(* Schneider Machine Expert - Basic project ECC, file version 2.0.0.0 *)
(* ProjectInformations: Name=New project *)

HARDWARE
  Cpu 0: TM221CE16T
  Cartridge1 0: TMC2SL1
  EthernetConfiguration: NetworkName=M221, IpAllocationMode=FixedAddress, IpAddress=192.168.1.10, SubnetMask=255.255.255.0
  EthernetConfiguration: NetworkName=M221, IpAllocationMode=FixedAddress, IpAddress=0.0.0.0, SubnetMask=0.0.0.0
  SerialLineConfiguration: Baud=Baud9600, Parity=ParityNone, DataBits=DataBits8, StopBits=StopBits1, PhysicalMedium=PhysicalMediumRs485, TransmissionMode=TransmissionModeModbusRtu, SlaveId=1, Addressing=MasterAddressing
  MastTask: UsePeriodScanMode=false, PeriodScan=100
  FastTask: Period=255
  CpuBehavior: StartingMode=StartAsPreviousState, AutoSaveRamOnEeprom=true, WatchdogPeriod=250

SYMBOLS  (address, symbol, comment, settings)
  %MW5:X2   BUZZER
  %MW5:X3   FLICKER
  %M100       "机械报警&蜂鸣器接口"
  %M103       "报警闪烁接口"
  %M110       "主机主滑油进口压力过低降速输出"
  %M111       "主机滑油进口温度过高降速输出"
  %M112       "主机十字头滑油进口压力过低降速输出"
  %M113       "主机推力轴承油温度过高降速输出"
  %M120       "主机增压器滑油进口压力过低降速输出"
  %M121       "主机增压器滑油出口温度过高降速输出"
  %M122       "主机缸套冷却水进口压力过低降速输出"
  %M129       "主机空气弹簧气源进口压力过低降速输出"
  %M130       "主机空冷器后扫气温度过高降速输出"
  %M131       "主机增压器前排气温度过高降速输出"
  %M132       "主机增压器后排气温度过高降速输出"
  %M200       "原先是%M100"
  %S5       SB_TB100MS  "内部时钟生成的 100 毫秒时基"
  %MW4        "通讯故障"
  %TM0        "可修改通讯间隔，默认10ms"  [Preset=10, Base=TenMilliSeconds]
  %TM1        [Preset=5, Base=OneHundredMilliSeconds]
  %TM2        [Preset=5, Base=OneHundredMilliSeconds]
  %TM3        [Preset=15, Base=OneSecond]
  %READ_VAR0   [Link(Value(FBComLinkParameterEnums=SerialLine1)), RemoteDeviceId(Value(int=1)), Timeout(Value(int=3)), ObjType(Value(FBComObjTypeParameterEnums=IW)), FirstObj(Value(int=513)), Quantity(Value(int=4)), IndexData(Value(int=0))]
  %WRITE_VAR0   [Link(Value(FBComLinkParameterEnums=SerialLine1)), RemoteDeviceId(Value(int=2)), Timeout(Value(int=3)), ObjType(Value(FBComObjTypeParameterEnums=MW)), FirstObj(Value(int=513)), Quantity(Value(int=2)), IndexData(Value(int=5))]
  %WRITE_VAR1   [Link(Value(FBComLinkParameterEnums=SerialLine1)), RemoteDeviceId(Value(int=3)), Timeout(Value(int=3)), ObjType(Value(FBComObjTypeParameterEnums=MW)), FirstObj(Value(int=513)), Quantity(Value(int=8)), IndexData(Value(int=10))]
  %WRITE_VAR2   [Link(Value(FBComLinkParameterEnums=SerialLine1)), RemoteDeviceId(Value(int=4)), Timeout(Value(int=3)), ObjType(Value(FBComObjTypeParameterEnums=MW)), FirstObj(Value(int=513)), Quantity(Value(int=8)), IndexData(Value(int=20))]
  %WRITE_VAR3   [Link(Value(FBComLinkParameterEnums=SerialLine1)), RemoteDeviceId(Value(int=5)), Timeout(Value(int=3)), ObjType(Value(FBComObjTypeParameterEnums=MW)), FirstObj(Value(int=513)), Quantity(Value(int=2)), IndexData(Value(int=30))]
  %WRITE_VAR4   [Link(Value(FBComLinkParameterEnums=SerialLine1)), RemoteDeviceId(Value(int=6)), Timeout(Value(int=3)), ObjType(Value(FBComObjTypeParameterEnums=SINGLE_REG)), FirstObj(Value(int=513)), Quantity(Value(int=1)), IndexData(Value(int=35))]

POU Communication
  (* SectionNumber=1 *)

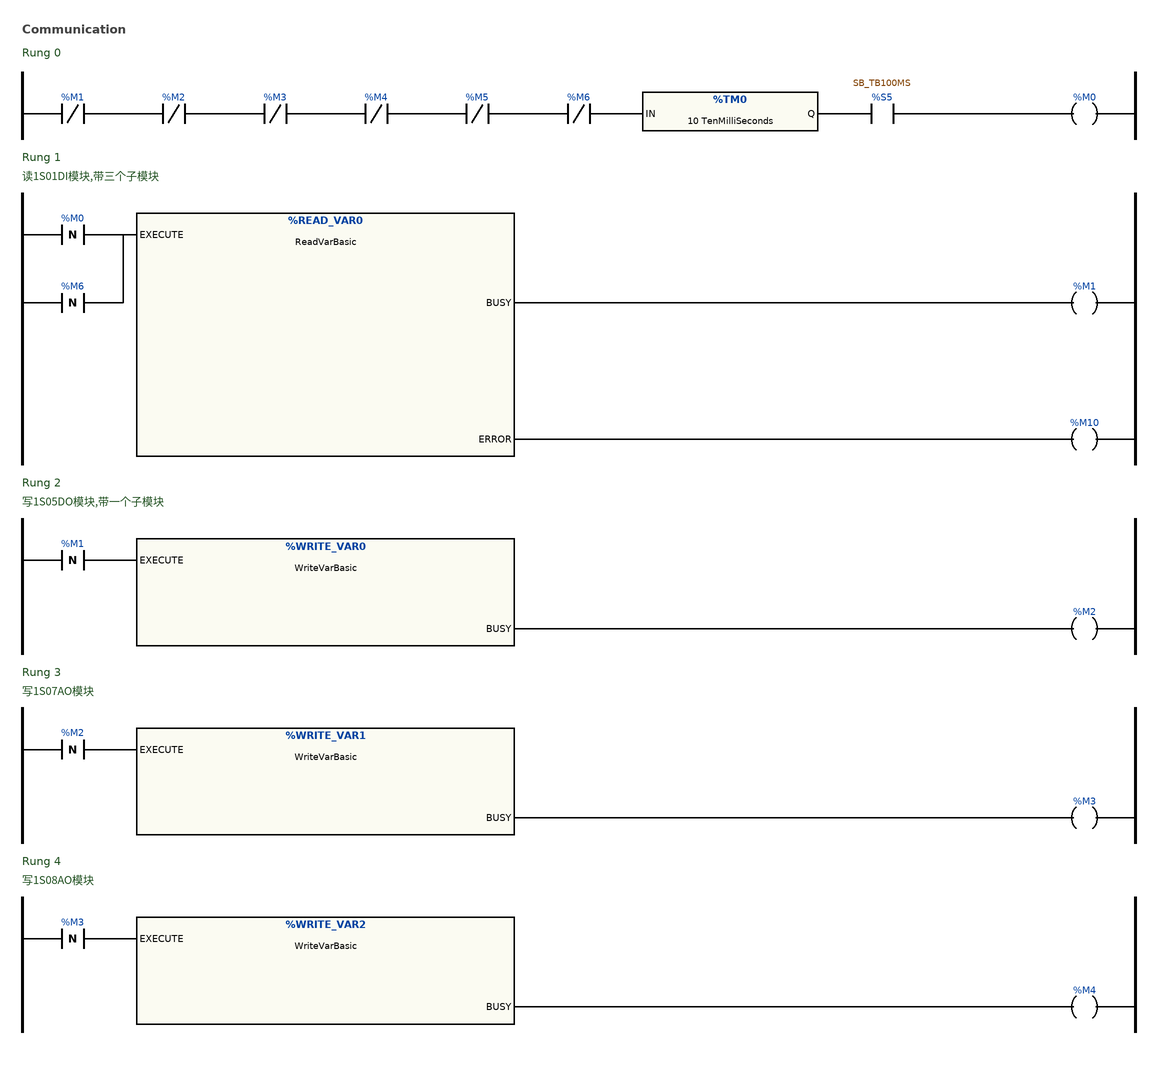

// Rung 0
  BLK %TM0
  LDN %M1
  ANDN %M2
  ANDN %M3
  ANDN %M4
  ANDN %M5
  ANDN %M6
  IN
  OUT_BLK
  LD Q
  AND %S5                 (* SB_TB100MS *)
  ST %M0
  END_BLK
  // as ST:
  //   %TM0(IN := NOT %M1 AND NOT %M2 AND NOT %M3 AND NOT %M4 AND NOT %M5 AND NOT %M6);
  //   %M0 := %TM0.Q AND SB_TB100MS;

// Rung 1
// 读1S01DI模块,带三个子模块
  BLK %READ_VAR0
  LDF %M0
  ORF %M6
  EXECUTE
  OUT_BLK
  LD BUSY
  ST %M1
  LD ERROR
  ST %M10
  END_BLK
  // as ST:
  //   %READ_VAR0(EXECUTE := FALLING(%M0) OR FALLING(%M6));
  //   %M1 := %READ_VAR0.BUSY;
  //   %M10 := %READ_VAR0.ERROR;

// Rung 2
// 写1S05DO模块,带一个子模块
  BLK %WRITE_VAR0
  LDF %M1
  EXECUTE
  OUT_BLK
  LD BUSY
  ST %M2
  END_BLK
  // as ST:
  //   %WRITE_VAR0(EXECUTE := FALLING(%M1));
  //   %M2 := %WRITE_VAR0.BUSY;

// Rung 3
// 写1S07AO模块
  BLK %WRITE_VAR1
  LDF %M2
  EXECUTE
  OUT_BLK
  LD BUSY
  ST %M3
  END_BLK
  // as ST:
  //   %WRITE_VAR1(EXECUTE := FALLING(%M2));
  //   %M3 := %WRITE_VAR1.BUSY;

// Rung 4
// 写1S08AO模块
  BLK %WRITE_VAR2
  LDF %M3
  EXECUTE
  OUT_BLK
  LD BUSY
  ST %M4
  END_BLK
  // as ST:
  //   %WRITE_VAR2(EXECUTE := FALLING(%M3));
  //   %M4 := %WRITE_VAR2.BUSY;

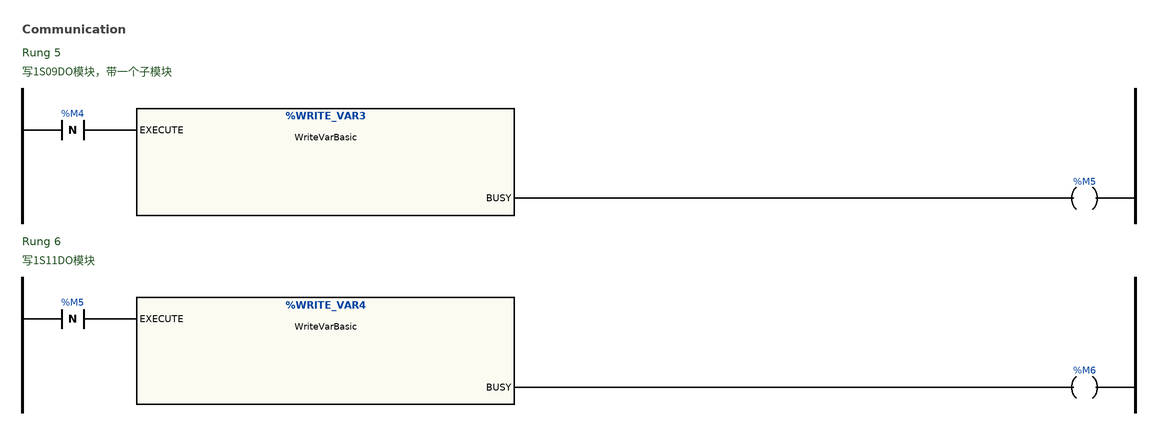

// Rung 5
// 写1S09DO模块，带一个子模块
  BLK %WRITE_VAR3
  LDF %M4
  EXECUTE
  OUT_BLK
  LD BUSY
  ST %M5
  END_BLK
  // as ST:
  //   %WRITE_VAR3(EXECUTE := FALLING(%M4));
  //   %M5 := %WRITE_VAR3.BUSY;

// Rung 6
// 写1S11DO模块
  BLK %WRITE_VAR4
  LDF %M5
  EXECUTE
  OUT_BLK
  LD BUSY
  ST %M6
  END_BLK
  // as ST:
  //   %WRITE_VAR4(EXECUTE := FALLING(%M5));
  //   %M6 := %WRITE_VAR4.BUSY;

POU Alarm&1S05&1SC01
  (* SectionNumber=2 *)

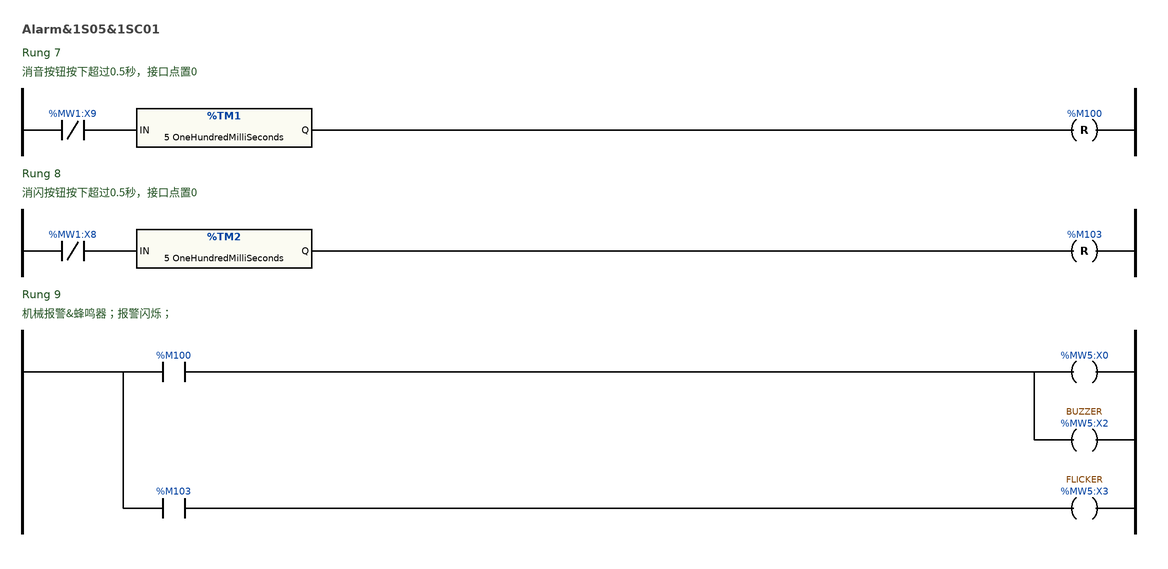

// Rung 7
// 消音按钮按下超过0.5秒，接口点置0
  BLK %TM1
  LDN %MW1:X9
  IN
  OUT_BLK
  LD Q
  R %M100
  END_BLK
  // as ST:
  //   %TM1(IN := NOT %MW1:X9);
  //   IF %TM1.Q THEN %M100 := FALSE; END_IF;

// Rung 8
// 消闪按钮按下超过0.5秒，接口点置0
  BLK %TM2
  LDN %MW1:X8
  IN
  OUT_BLK
  LD Q
  R %M103
  END_BLK
  // as ST:
  //   %TM2(IN := NOT %MW1:X8);
  //   IF %TM2.Q THEN %M103 := FALSE; END_IF;

// Rung 9
// 机械报警&蜂鸣器；报警闪烁；
  LD 1
  MPS
  AND %M100
  ST %MW5:X0
  ST %MW5:X2
  MPP
  AND %M103
  ST %MW5:X3
  // as ST:
  //   %MW5:X0 := %M100;
  //   %MW5:X2 := %M100;
  //   %MW5:X3 := %M103;

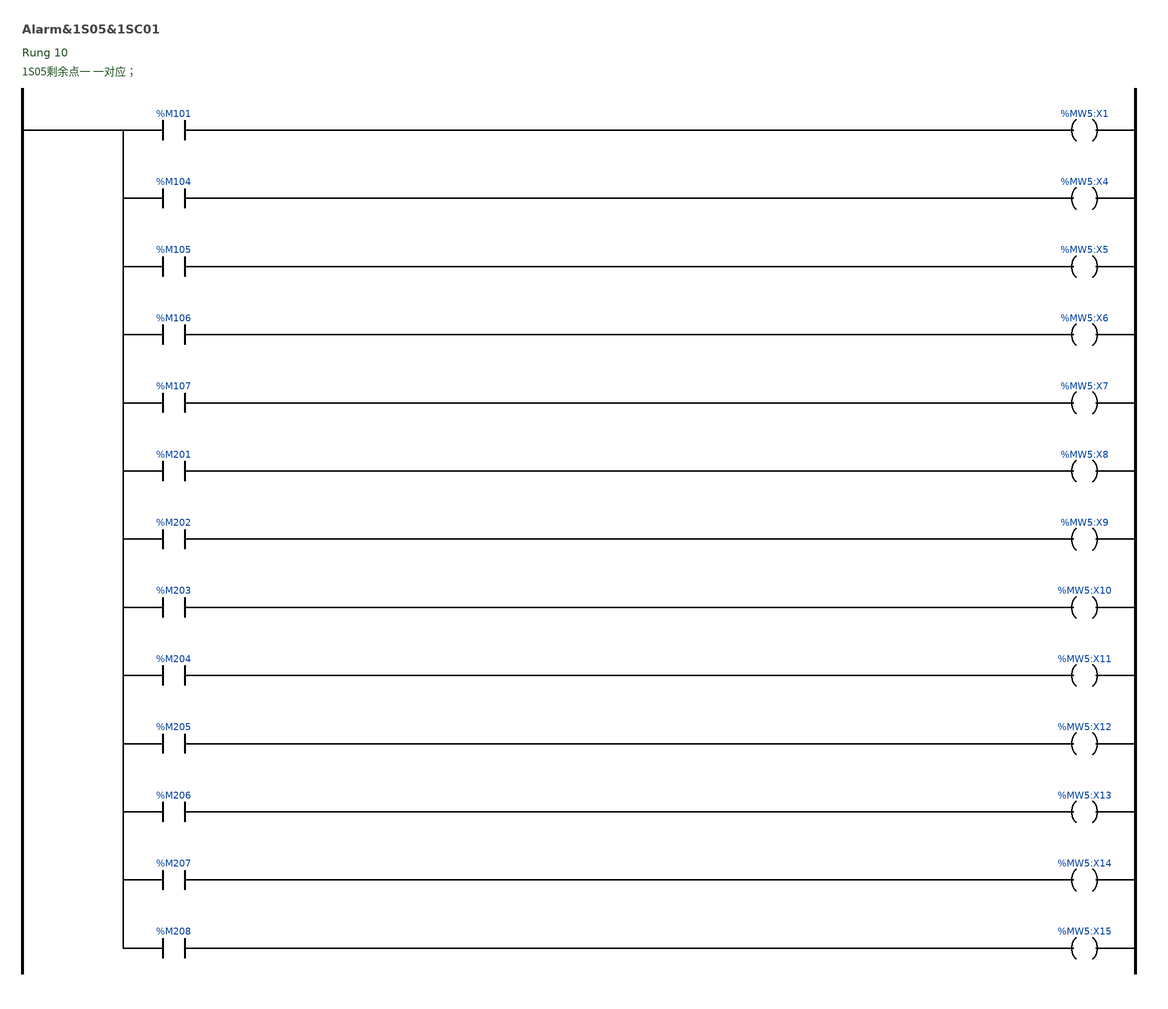

// Rung 10
// 1S05剩余点一 一对应；
  LD 1
  MPS
  AND %M101
  ST %MW5:X1
  MRD
  AND %M104
  ST %MW5:X4
  MRD
  AND %M105
  ST %MW5:X5
  MRD
  AND %M106
  ST %MW5:X6
  MRD
  AND %M107
  ST %MW5:X7
  MRD
  AND %M201
  ST %MW5:X8
  MRD
  AND %M202
  ST %MW5:X9
  MRD
  AND %M203
  ST %MW5:X10
  MRD
  AND %M204
  ST %MW5:X11
  MRD
  AND %M205
  ST %MW5:X12
  MRD
  AND %M206
  ST %MW5:X13
  MRD
  AND %M207
  ST %MW5:X14
  MPP
  AND %M208
  ST %MW5:X15
  // as ST:
  //   %MW5:X1 := %M101;
  //   %MW5:X4 := %M104;
  //   %MW5:X5 := %M105;
  //   %MW5:X6 := %M106;
  //   %MW5:X7 := %M107;
  //   %MW5:X8 := %M201;
  //   %MW5:X9 := %M202;
  //   %MW5:X10 := %M203;
  //   %MW5:X11 := %M204;
  //   %MW5:X12 := %M205;
  //   %MW5:X13 := %M206;
  //   %MW5:X14 := %M207;
  //   %MW5:X15 := %M208;

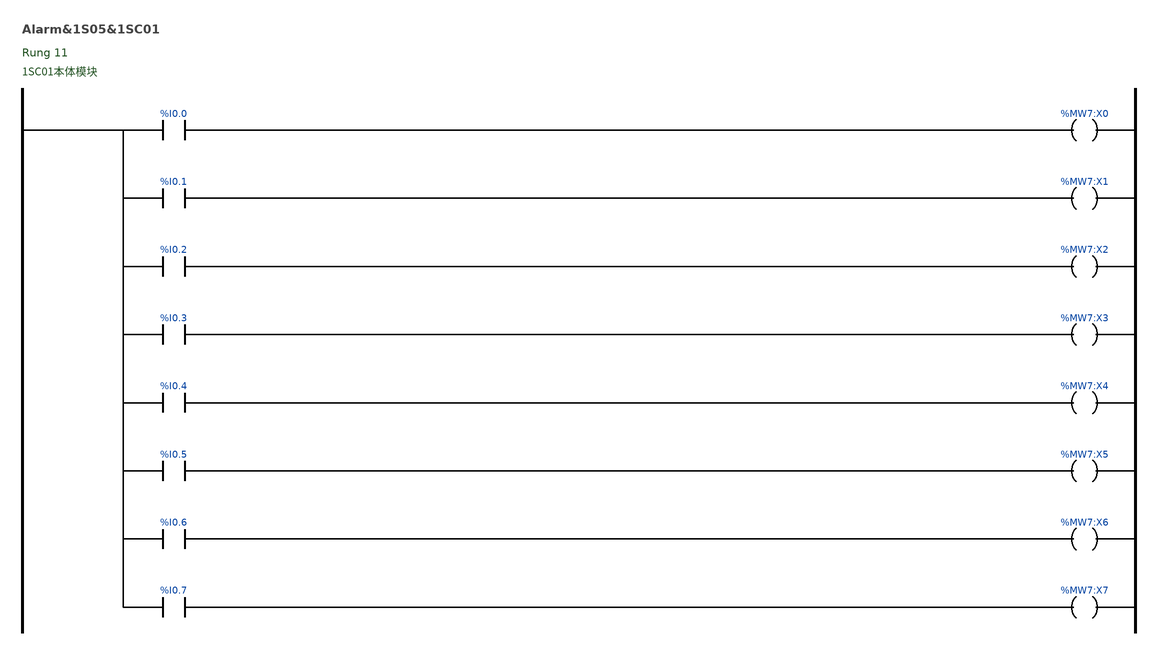

// Rung 11
// 1SC01本体模块
  LD 1
  MPS
  AND %I0.0
  ST %MW7:X0
  MRD
  AND %I0.1
  ST %MW7:X1
  MRD
  AND %I0.2
  ST %MW7:X2
  MRD
  AND %I0.3
  ST %MW7:X3
  MRD
  AND %I0.4
  ST %MW7:X4
  MRD
  AND %I0.5
  ST %MW7:X5
  MRD
  AND %I0.6
  ST %MW7:X6
  MPP
  AND %I0.7
  ST %MW7:X7
  // as ST:
  //   %MW7:X0 := %I0.0;
  //   %MW7:X1 := %I0.1;
  //   %MW7:X2 := %I0.2;
  //   %MW7:X3 := %I0.3;
  //   %MW7:X4 := %I0.4;
  //   %MW7:X5 := %I0.5;
  //   %MW7:X6 := %I0.6;
  //   %MW7:X7 := %I0.7;

POU CommError
  (* SectionNumber=3 *)

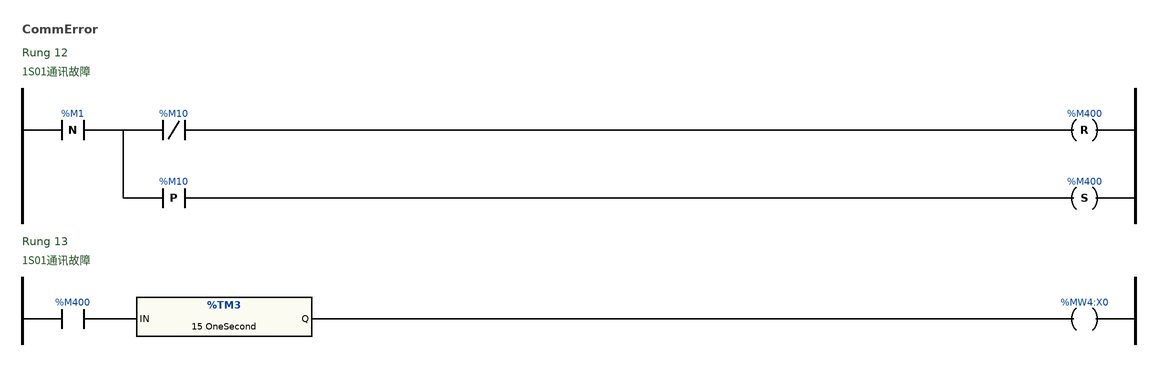

// Rung 12
// 1S01通讯故障
  LDF %M1
  MPS
  ANDN %M10
  R %M400
  MPP
  ANDR %M10
  S %M400
  // as ST:
  //   IF FALLING(%M1) AND NOT %M10 THEN %M400 := FALSE; END_IF;
  //   IF FALLING(%M1) AND RISING(%M10) THEN %M400 := TRUE; END_IF;

// Rung 13
// 1S01通讯故障
  BLK %TM3
  LD %M400
  IN
  OUT_BLK
  LD Q
  ST %MW4:X0
  END_BLK
  // as ST:
  //   %TM3(IN := %M400);
  //   %MW4:X0 := %TM3.Q;

POU SlowDown&1S11
  (* SectionNumber=4 *)

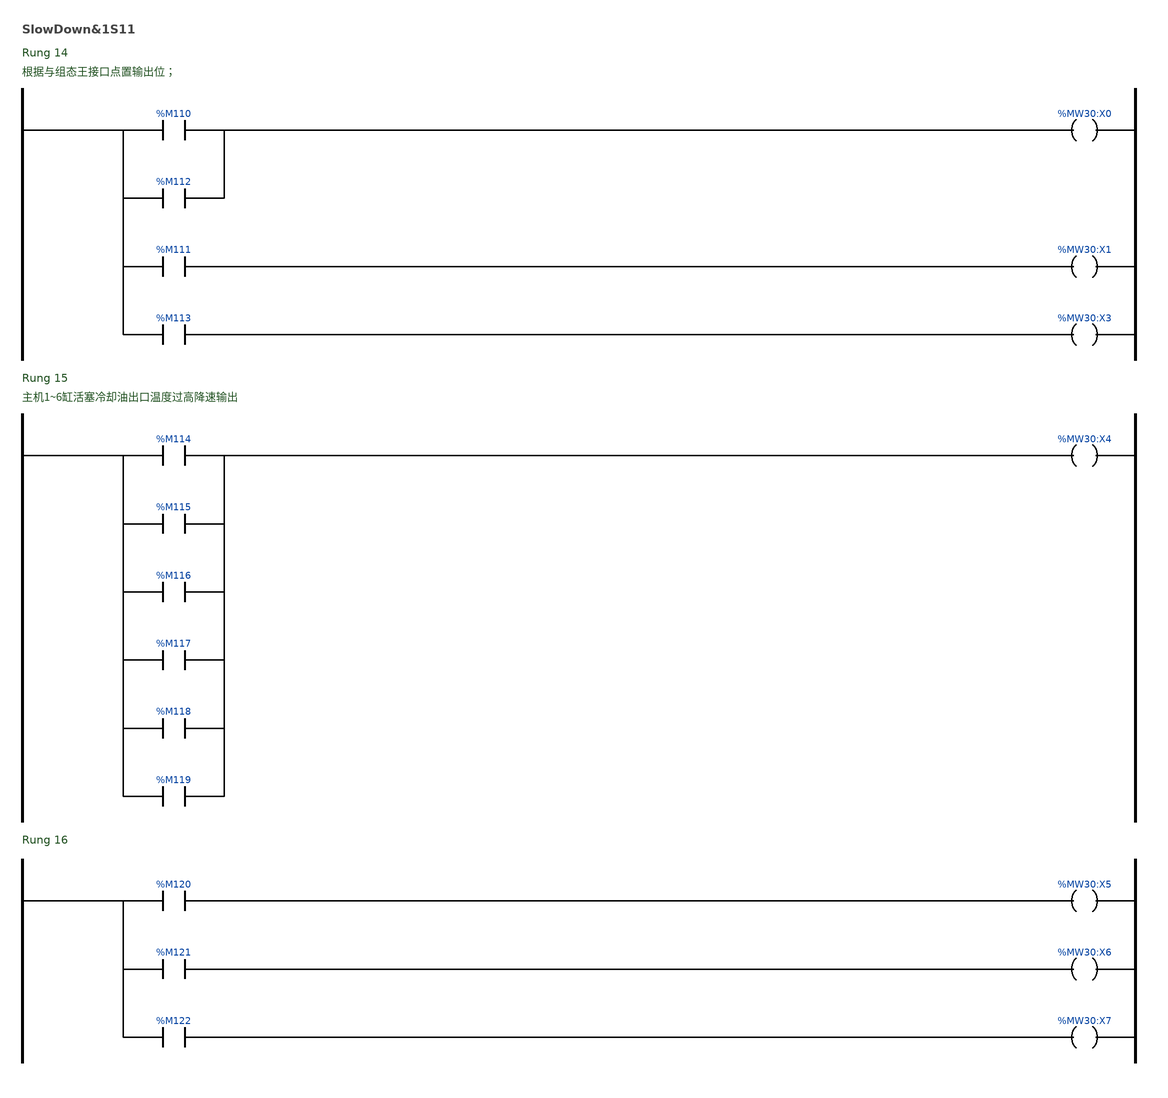

// Rung 14
// 根据与组态王接口点置输出位；
  LD 1
  MPS
  AND( %M110
  OR %M112
  )
  ST %MW30:X0
  MRD
  AND %M111
  ST %MW30:X1
  MPP
  AND %M113
  ST %MW30:X3
  // as ST:
  //   %MW30:X0 := %M110 OR %M112;
  //   %MW30:X1 := %M111;
  //   %MW30:X3 := %M113;

// Rung 15
// 主机1~6缸活塞冷却油出口温度过高降速输出
  LD 1
  AND( %M114
  OR %M115
  OR %M116
  OR %M117
  OR %M118
  OR %M119
  )
  ST %MW30:X4
  // as ST:
  //   %MW30:X4 := %M114 OR %M115 OR %M116 OR %M117 OR %M118 OR %M119;

// Rung 16
  LD 1
  MPS
  AND %M120
  ST %MW30:X5
  MRD
  AND %M121
  ST %MW30:X6
  MPP
  AND %M122
  ST %MW30:X7
  // as ST:
  //   %MW30:X5 := %M120;
  //   %MW30:X6 := %M121;
  //   %MW30:X7 := %M122;

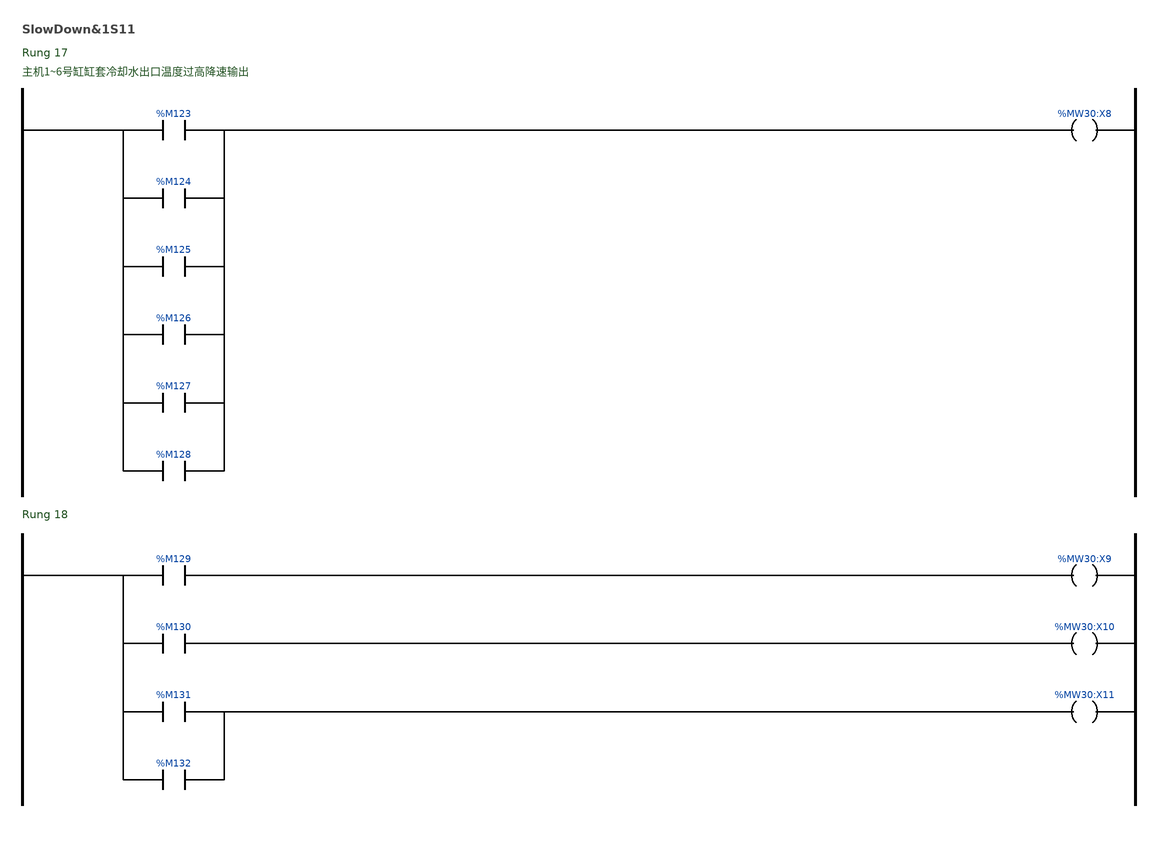

// Rung 17
// 主机1~6号缸缸套冷却水出口温度过高降速输出
  LD 1
  AND( %M123
  OR %M124
  OR %M125
  OR %M126
  OR %M127
  OR %M128
  )
  ST %MW30:X8
  // as ST:
  //   %MW30:X8 := %M123 OR %M124 OR %M125 OR %M126 OR %M127 OR %M128;

// Rung 18
  LD 1
  MPS
  AND %M129
  ST %MW30:X9
  MRD
  AND %M130
  ST %MW30:X10
  MPP
  AND( %M131
  OR %M132
  )
  ST %MW30:X11
  // as ST:
  //   %MW30:X9 := %M129;
  //   %MW30:X10 := %M130;
  //   %MW30:X11 := %M131 OR %M132;

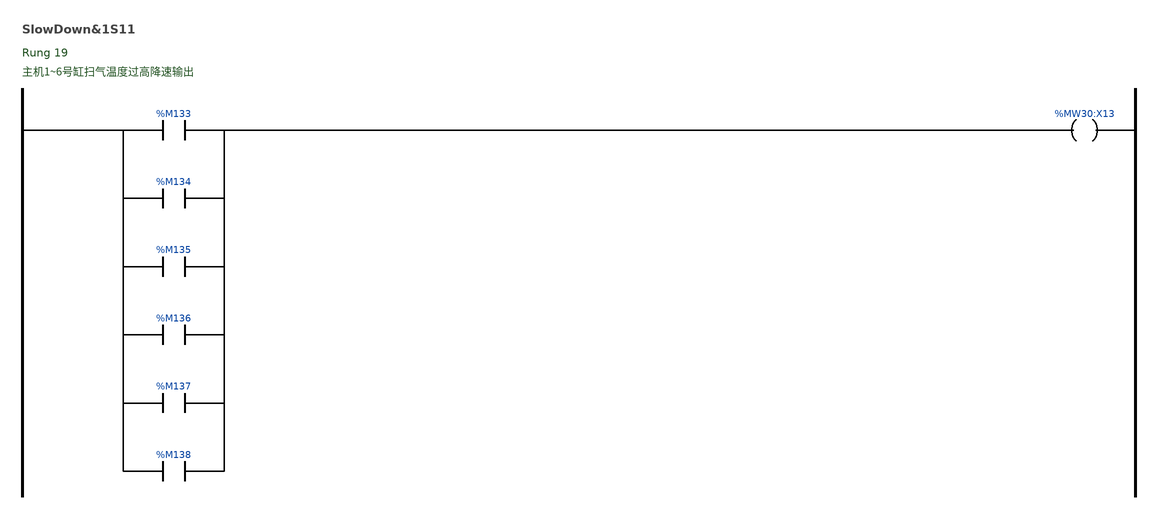

// Rung 19
// 主机1~6号缸扫气温度过高降速输出
  LD 1
  AND( %M133
  OR %M134
  OR %M135
  OR %M136
  OR %M137
  OR %M138
  )
  ST %MW30:X13
  // as ST:
  //   %MW30:X13 := %M133 OR %M134 OR %M135 OR %M136 OR %M137 OR %M138;

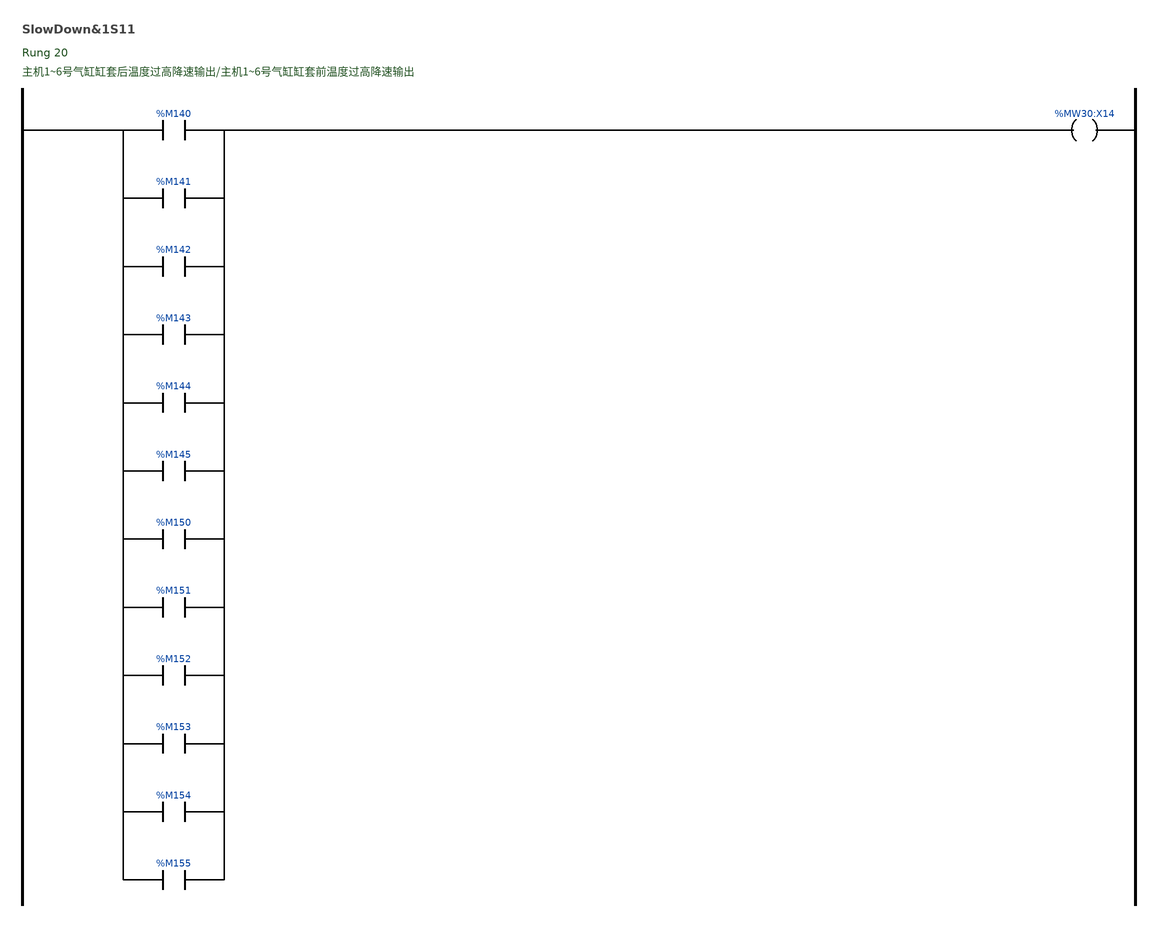

// Rung 20
// 主机1~6号气缸缸套后温度过高降速输出/主机1~6号气缸缸套前温度过高降速输出
  LD 1
  AND( %M140
  OR %M141
  OR %M142
  OR %M143
  OR %M144
  OR %M145
  OR %M150
  OR %M151
  OR %M152
  OR %M153
  OR %M154
  OR %M155
  )
  ST %MW30:X14
  // as ST:
  //   %MW30:X14 := %M140 OR %M141 OR %M142 OR %M143 OR %M144 OR %M145 OR %M150 OR %M151 OR %M152 OR %M153 OR %M154 OR %M155;

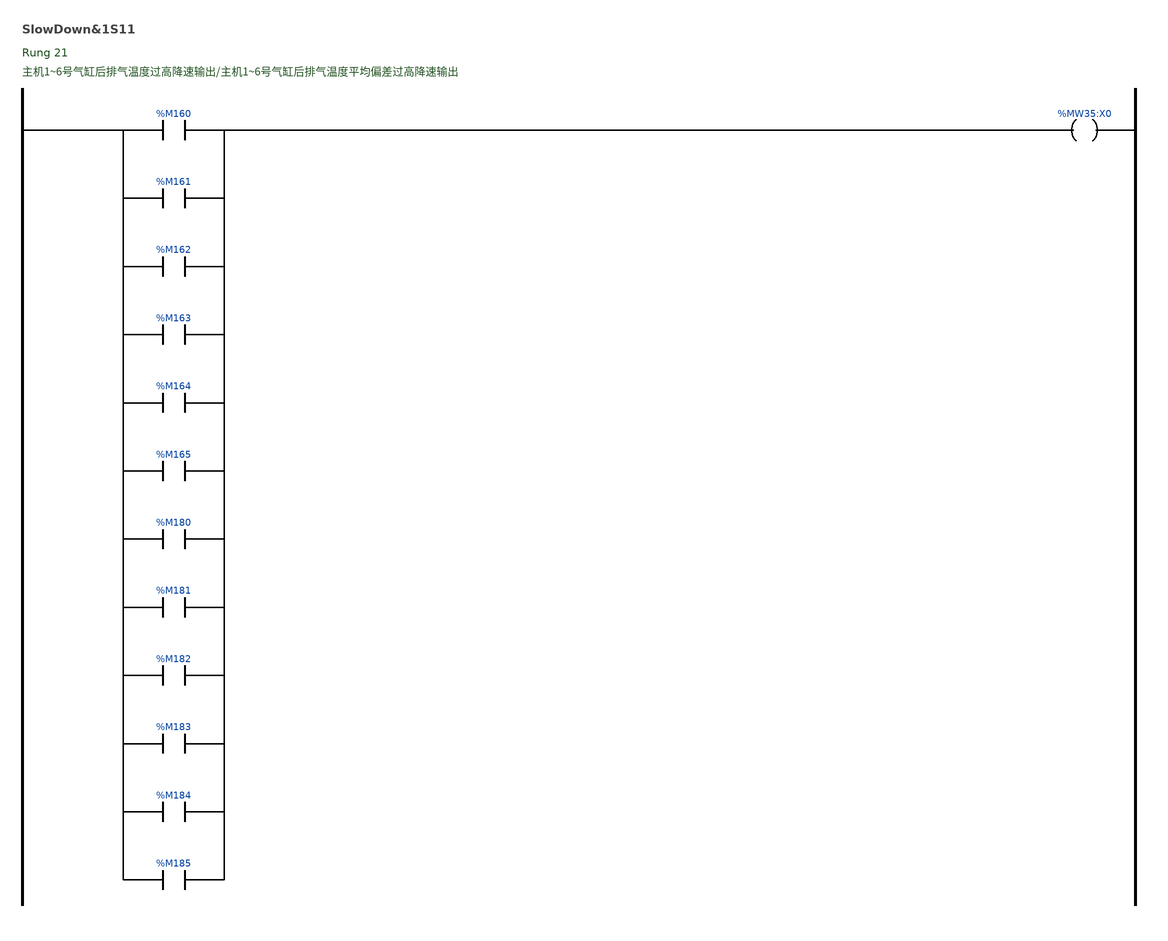

// Rung 21
// 主机1~6号气缸后排气温度过高降速输出/主机1~6号气缸后排气温度平均偏差过高降速输出
  LD 1
  AND( %M160
  OR %M161
  OR %M162
  OR %M163
  OR %M164
  OR %M165
  OR %M180
  OR %M181
  OR %M182
  OR %M183
  OR %M184
  OR %M185
  )
  ST %MW35:X0
  // as ST:
  //   %MW35:X0 := %M160 OR %M161 OR %M162 OR %M163 OR %M164 OR %M165 OR %M180 OR %M181 OR %M182 OR %M183 OR %M184 OR %M185;

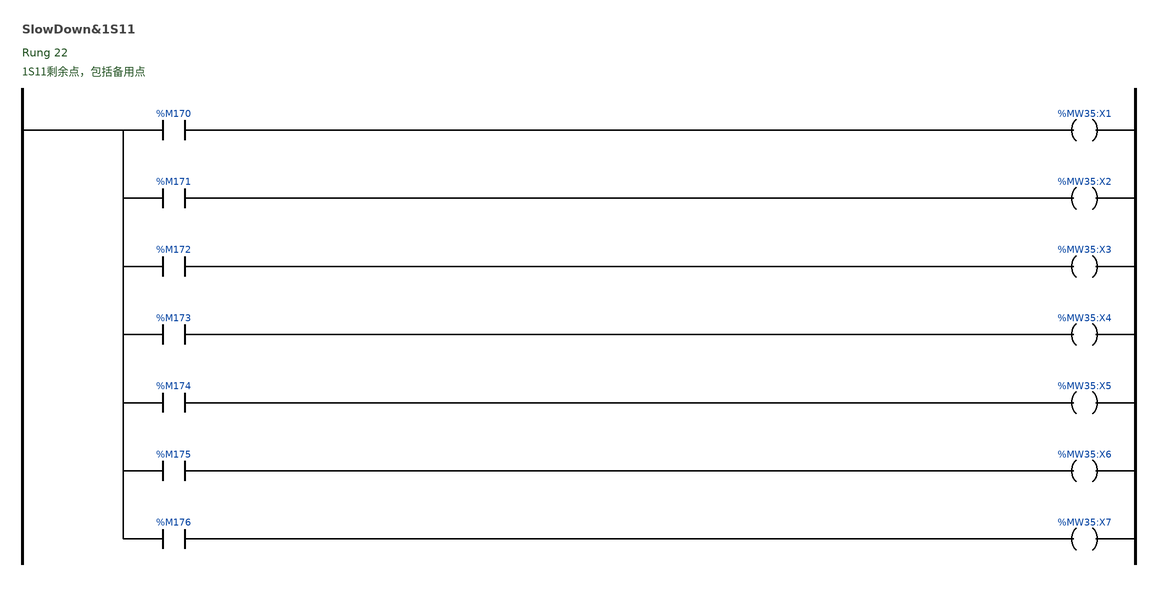

// Rung 22
// 1S11剩余点，包括备用点
  LD 1
  MPS
  AND %M170
  ST %MW35:X1
  MRD
  AND %M171
  ST %MW35:X2
  MRD
  AND %M172
  ST %MW35:X3
  MRD
  AND %M173
  ST %MW35:X4
  MRD
  AND %M174
  ST %MW35:X5
  MRD
  AND %M175
  ST %MW35:X6
  MPP
  AND %M176
  ST %MW35:X7
  // as ST:
  //   %MW35:X1 := %M170;
  //   %MW35:X2 := %M171;
  //   %MW35:X3 := %M172;
  //   %MW35:X4 := %M173;
  //   %MW35:X5 := %M174;
  //   %MW35:X6 := %M175;
  //   %MW35:X7 := %M176;
